FUNCTION Convert_DWORD_TO_UINT : Hresult
VAR_INPUT
	in : DWORD;
	out : REFERENCE TO UINT;
END_VAR
VAR
	converted : UINT;
END_VAR

converted := DWORD_TO_UINT(in);

IF (UINT_TO_DWORD(converted) <> in) THEN
	Convert_DWORD_TO_UINT := INCOMPATIBLE;
	RETURN;
END_IF

out := converted;

END_FUNCTION

(* stored: Version 1.1.0.1, ProductVersion 3.1.4024.12
   POU Convert_DWORD_TO_UINT: Id {95b1d7f8-e3c7-4143-a910-0350e743a662}, SpecialFunc None *)
